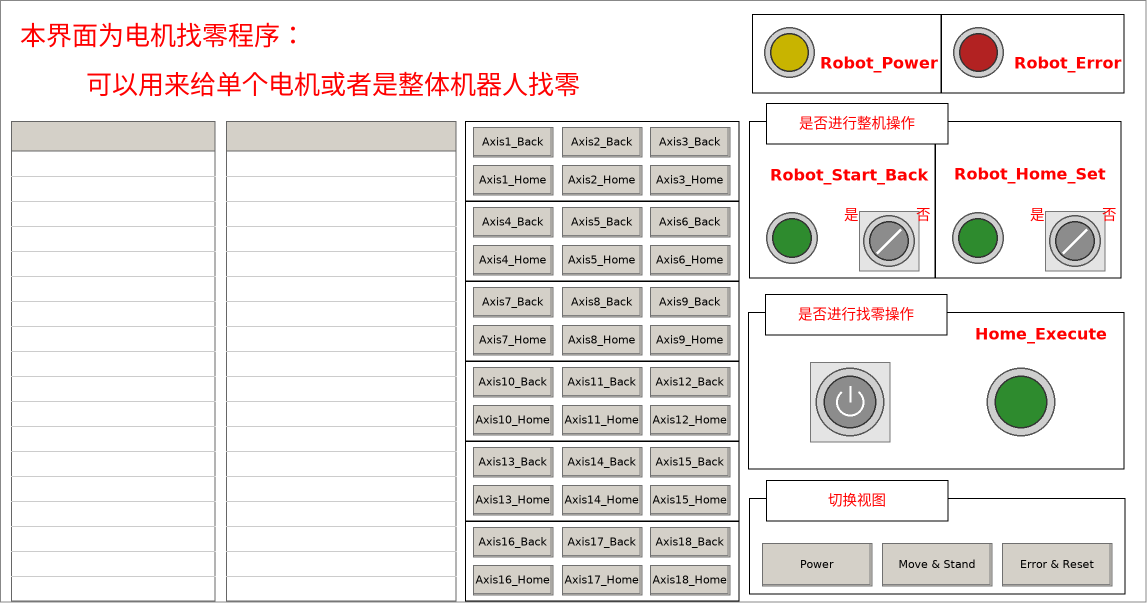
VISUALIZATION Visu_Home  // 1147x603
    Rectangle (752,14 189x79)
    Rectangle (748,312 376x157)
    Label (964,318 154x32), "Home_Execute"
    Rectangle (765,294 182x41), "是否进行找零操作"
    Lamp1 (981,362 80x80), variable: MAIN.Home_Execute, style: Lamp-Lamp1-Green
    PowerSwitch (810,362 80x80), variable: MAIN.Home_Execute, behaviour: TOGGLE, style: Switch-PowerSwitch-Gray
    Rectangle (941,14 183x79)
    Lamp1 (948,23 61x59), variable: MAIN.Robot_Error, style: Lamp-Lamp1-Red
    Label (991,47 154x32), "Robot_Error"
    Label (17,15 365x42), "本界面为电机找零程序："
    Label (83,64 874x42), "可以用来给单个电机或者是整体机器人找零"
    Table (11,121 204x480), data array: MAIN.Axis_ActPostion
        p3854506369: MAIN.Axis_ActPostion[INDEX]
    Table (226,121 230x480), data array: MAIN.Current_Turque_Value
        p3854506369: MAIN.Current_Turque_Value[INDEX]
    Lamp1 (759,23 61x59), variable: MAIN.Robot_Power, style: Lamp-Lamp1-Yellow
    Label (802,47 154x32), "Robot_Power"
    Rectangle (465,121 274x80)
    Button (473,127 80x30), "Axis1_Back"
        toggle MAIN.Axis_Start_Back[1]
        OnMouseClick: change screen: Visu_Home
    Button (473,165 80x30), "Axis1_Home"
        tap MAIN.Axis_Home_Set[1]
        OnMouseClick: change screen: Visu_Home
    Button (650,127 80x30), "Axis3_Back"
        toggle MAIN.Axis_Start_Back[3]
        OnMouseClick: change screen: Visu_Home
    Button (650,165 80x30), "Axis3_Home"
        tap MAIN.Axis_Home_Set[3]
        OnMouseClick: change screen: Visu_Home
    Button (562,127 80x30), "Axis2_Back"
        toggle MAIN.Axis_Start_Back[2]
        OnMouseClick: change screen: Visu_Home
    Button (562,165 80x30), "Axis2_Home"
        tap MAIN.Axis_Home_Set[2]
        OnMouseClick: change screen: Visu_Home
    Rectangle (465,201 274x80)
    Button (473,207 80x30), "Axis4_Back"
        toggle MAIN.Axis_Start_Back[4]
        OnMouseClick: change screen: Visu_Home
    Button (473,245 80x30), "Axis4_Home"
        tap MAIN.Axis_Home_Set[4]
        OnMouseClick: change screen: Visu_Home
    Button (650,207 80x30), "Axis6_Back"
        toggle MAIN.Axis_Start_Back[6]
        OnMouseClick: change screen: Visu_Home
    Button (650,245 80x30), "Axis6_Home"
        tap MAIN.Axis_Home_Set[6]
        OnMouseClick: change screen: Visu_Home
    Button (562,207 80x30), "Axis5_Back"
        toggle MAIN.Axis_Start_Back[5]
        OnMouseClick: change screen: Visu_Home
    Button (562,245 80x30), "Axis5_Home"
        tap MAIN.Axis_Home_Set[5]
        OnMouseClick: change screen: Visu_Home
    Rectangle (465,281 274x80)
    Button (473,287 80x30), "Axis7_Back"
        toggle MAIN.Axis_Start_Back[7]
        OnMouseClick: change screen: Visu_Home
    Button (473,325 80x30), "Axis7_Home"
        tap MAIN.Axis_Home_Set[7]
        OnMouseClick: change screen: Visu_Home
    Button (650,287 80x30), "Axis9_Back"
        toggle MAIN.Axis_Start_Back[9]
        OnMouseClick: change screen: Visu_Home
    Button (650,325 80x30), "Axis9_Home"
        tap MAIN.Axis_Home_Set[9]
        OnMouseClick: change screen: Visu_Home
    Button (562,287 80x30), "Axis8_Back"
        toggle MAIN.Axis_Start_Back[8]
        OnMouseClick: change screen: Visu_Home
    Button (562,325 80x30), "Axis8_Home"
        tap MAIN.Axis_Home_Set[8]
        OnMouseClick: change screen: Visu_Home
    Rectangle (465,361 274x80)
    Button (473,367 80x30), "Axis10_Back"
        toggle MAIN.Axis_Start_Back[10]
        OnMouseClick: change screen: Visu_Home
    Button (473,405 80x30), "Axis10_Home"
        tap MAIN.Axis_Home_Set[10]
        OnMouseClick: change screen: Visu_Home
    Button (650,367 80x30), "Axis12_Back"
        toggle MAIN.Axis_Start_Back[12]
        OnMouseClick: change screen: Visu_Home
    Button (650,405 80x30), "Axis12_Home"
        tap MAIN.Axis_Home_Set[12]
        OnMouseClick: change screen: Visu_Home
    Button (562,367 80x30), "Axis11_Back"
        toggle MAIN.Axis_Start_Back[11]
        OnMouseClick: change screen: Visu_Home
    Button (562,405 80x30), "Axis11_Home"
        tap MAIN.Axis_Home_Set[11]
        OnMouseClick: change screen: Visu_Home
    Rectangle (465,441 274x80)
    Button (473,447 80x30), "Axis13_Back"
        toggle MAIN.Axis_Start_Back[13]
        OnMouseClick: change screen: Visu_Home
    Button (473,485 80x30), "Axis13_Home"
        tap MAIN.Axis_Home_Set[13]
        OnMouseClick: change screen: Visu_Home
    Button (650,447 80x30), "Axis15_Back"
        toggle MAIN.Axis_Start_Back[15]
        OnMouseClick: change screen: Visu_Home
    Button (650,485 80x30), "Axis15_Home"
        tap MAIN.Axis_Home_Set[15]
        OnMouseClick: change screen: Visu_Home
    Button (562,447 80x30), "Axis14_Back"
        toggle MAIN.Axis_Start_Back[14]
        OnMouseClick: change screen: Visu_Home
    Button (562,485 80x30), "Axis14_Home"
        tap MAIN.Axis_Home_Set[14]
        OnMouseClick: change screen: Visu_Home
    Rectangle (465,521 274x80)
    Button (473,527 80x30), "Axis16_Back"
        toggle MAIN.Axis_Start_Back[16]
        OnMouseClick: change screen: Visu_Home
    Button (473,565 80x30), "Axis16_Home"
        tap MAIN.Axis_Home_Set[16]
        OnMouseClick: change screen: Visu_Home
    Button (650,527 80x30), "Axis18_Back"
        toggle MAIN.Axis_Start_Back[18]
        OnMouseClick: change screen: Visu_Home
    Button (650,565 80x30), "Axis18_Home"
        tap MAIN.Axis_Home_Set[18]
        OnMouseClick: change screen: Visu_Home
    Button (562,527 80x30), "Axis17_Back"
        toggle MAIN.Axis_Start_Back[17]
        OnMouseClick: change screen: Visu_Home
    Button (562,565 80x30), "Axis17_Home"
        tap MAIN.Axis_Home_Set[17]
        OnMouseClick: change screen: Visu_Home
    Rectangle (935,121 186x157)
    Rectangle (749,121 186x157)
    Label (772,159 154x32), "Robot_Start_Back"
    Rectangle (766,103 182x41), "是否进行整机操作"
    Lamp1 (762,208 60x60), variable: MAIN.Robot_Start_Back, style: Lamp-Lamp1-Green
    RotarySwitch (859,209 60x64), variable: MAIN.Robot_Start_Back, behaviour: TOGGLE, style: Switch-RotarySwitch-Gray
    Label (901,203 45x24), "否"
    Label (829,203 45x24), "是"
    Lamp1 (948,208 60x60), variable: MAIN.Robot_Home_Set, style: Lamp-Lamp1-Green
    RotarySwitch (1045,209 60x64), variable: MAIN.Robot_Home_Set, behaviour: TOGGLE, style: Switch-RotarySwitch-Gray
    Label (1087,203 45x24), "否"
    Label (1015,203 45x24), "是"
    Label (953,158 154x32), "Robot_Home_Set"
    Group (749,480 376x114)
        Rectangle (0,18 376x96)
        Rectangle (17,0 182x41), "切换视图"
        Button (13,63 110x43), "Power"
            OnMouseClick: change screen: Visu_Power
        Button (253,63 110x43), "Error & Reset"
            OnMouseClick: change screen: Visu_Reset
        Button (133,63 110x43), "Move & Stand"
            OnMouseClick: change screen: Visu_Stand
END_VISUALIZATION

(* stored: Version 1.1.0.1, ProductVersion 3.1.4020.12
   Visu Visu_Home: Id {f1fd6469-4ee4-4390-8668-28dd879e70aa} *)
